// TIA Portal project "Project1-6-2" (V15.1)

(* hardware
DEVICE "S7300/ET200M station_1"  S7-300 station
   slot 0: "Rail_0"  Rail  6ES7 390-1***0-0AA0
   slot 2: "PLC_1"  CPU 313C-2 DP  6ES7 313-6CF03-0AB0  V2.6
      slot 0: "MPI interface_1"  X1
      slot 1: "DP interface_1"  X2
      slot 2: "DI 16/DO 16_1"  DI16/DO16
      slot 4: "Count_1"  Counter
*)

// ===== PLC "PLC_1"  CPU 313C-2 DP =====

VAR_GLOBAL   // PLC tag table "Default tag table"
   "Start" AT %I0.0 : Bool;
   "Stop" AT %I0.1 : Bool;
   "Tag_1" AT %M0.0 : Bool;
   "Tag_2" AT %M0.3 : Bool;
   "Counter" AT %C0 : Counter;
   "Tag_3" AT %MW2 : Word;
   "Timer" AT %T0 : Timer;
   "Working Robot" AT %Q0.0 : Bool;
   "Tag_4" AT %M0.1 : Bool;
   "Start 2" AT %M0.2 : Bool;
   "Tag_5" AT %M0.4 : Bool;
   "Memory Clock 0.5s" AT %M20.3 : Bool;
END_VAR

ORGANIZATION_BLOCK "Main"   // OB1, LAD
TITLE = "Main Program Sweep (Cycle)"
{ S7_Optimized_Access := 'FALSE' }
VERSION : 0.1
   VAR_TEMP
      OB1_EV_CLASS : Byte;   // Bits 0-3 = 1 (Coming event), Bits 4-7 = 1 (Event class 1)
      OB1_SCAN_1 : Byte;   // 1 (Cold restart scan 1 of OB 1), 3 (Scan 2-n of OB 1)
      OB1_PRIORITY : Byte;   // Priority of OB Execution
      OB1_OB_NUMBR : Byte;   // 1 (Organization block 1, OB1)
      OB1_RESERVED_1 : Byte;   // Reserved for system
      OB1_RESERVED_2 : Byte;   // Reserved for system
      OB1_PREV_CYCLE : Int;   // Cycle time of previous OB1 scan (milliseconds)
      OB1_MIN_CYCLE : Int;   // Minimum cycle time of OB1 (milliseconds)
      OB1_MAX_CYCLE : Int;   // Maximum cycle time of OB1 (milliseconds)
      OB1_DATE_TIME : Date_And_Time;   // Date and time OB1 started
   END_VAR
   VAR_TEMP   // added for the SCL form of the ladder/FBD networks
      _w1 : Bool;
      _s5time1 : S5Time;
   END_VAR
BEGIN

REGION Network 1
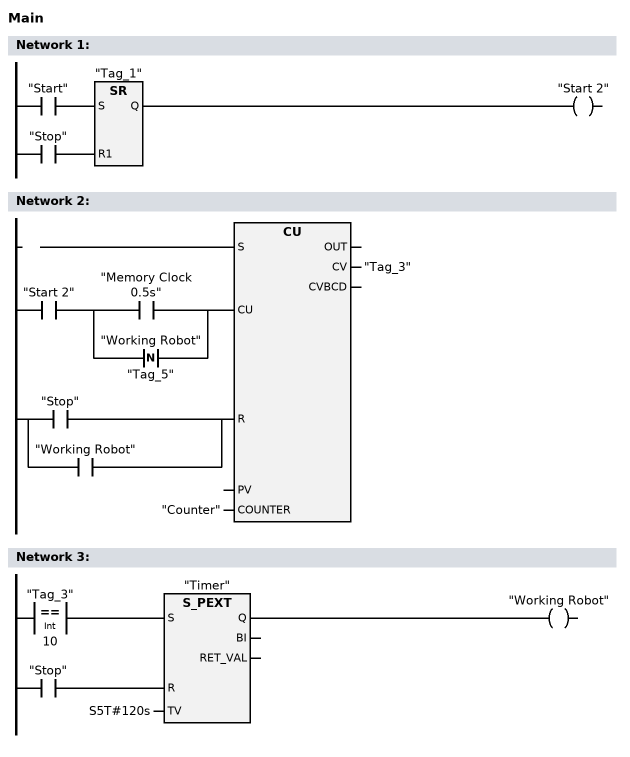
   RUNG wire#powerrail
      Contact( "Start" )
      S_SR(operand := "Tag_1", r1 := wire#w1)
      Coil( "Start 2" )
   END_RUNG
   RUNG wire#powerrail
      Contact( "Stop" )
   END_RUNG wire#w1
   // the same network as SCL:
   IF "Start" THEN
       "Tag_1" := TRUE;   // SR flip-flop
   END_IF;
   IF "Stop" THEN "Tag_1" := FALSE; END_IF;
   "Start 2" := "Tag_1";
END_REGION

REGION Network 2
   // no SCL statement known for Cu: written as a call
   #_w1 := "Start 2" AND NOT "Working Robot" AND "Tag_5";   // falling edge of "Working Robot"
   "Tag_5" := "Working Robot";
   Cu(cu := ("Start 2" AND "Memory Clock 0.5s") OR #_w1,
      r := "Stop" OR "Working Robot",
      "counter" := "Counter",
      cv => "Tag_3");
END_REGION

REGION Network 3
   RUNG wire#powerrail
      { S7_Templates := "SrcType := Int" } EQ_Contact(in1 := "Tag_3", in2 := 10)
      S_PEXT(T_NO := "Timer", R := wire#w1, TV := S5T#120s, BI =>, RET_VAL =>)
      Coil( "Working Robot" )
   END_RUNG
   RUNG wire#powerrail
      Contact( "Stop" )
   END_RUNG wire#w1
   // the same network as SCL:
   #_s5time1 := S_PEXT(T_NO := "Timer", S := "Tag_3" = 10, R := "Stop", TV := S5T#120s, Q => #_w1);
   "Working Robot" := #_w1;
END_REGION
END_ORGANIZATION_BLOCK